// LS Electric XG5000 project: XBM_MODBUS
// PLC NewPLC
// module base 0 slot 0: 입출력 모듈:XBM-DN32H (DC 24V입력/TR 출력, 32점)
// module base 0 slot 2: 아날로그입출력 모듈:XBF-AH04A (A/D 전압/전류 2채널, D/A 전압/전류 2채널)

PROGRAM NewProgram (task: 스캔 프로그램)

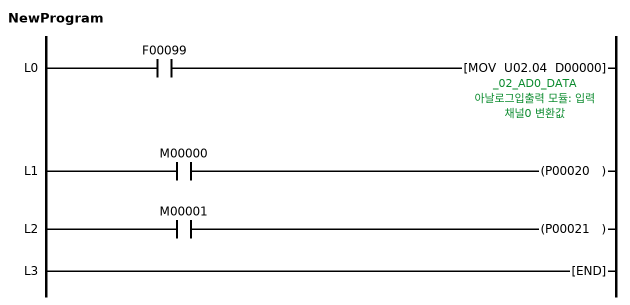
; L0
LOAD      F00099
MOV       U02.04 D00000	// _02_AD0_DATA 아날로그입출력 모듈: 입력 채널0 변환값
; L1
LOAD      M00000
OUT       P00020
; L2
LOAD      M00001
OUT       P00021
; L3
END